FUNCTION_BLOCK FB_Base
VAR_INPUT
END_VAR
VAR_OUTPUT
END_VAR
VAR
	_CalcCounter : INT;
END_VAR

{attribute 'monitoring' := 'call'}
PROPERTY CalcCounter : INT
GET
CalcCounter := _CalcCounter;
END_GET
SET
_CalcCounter := CalcCounter;
END_SET
END_PROPERTY

{attribute 'TcRpcEnable'}
METHOD Calculation : REAL
VAR_INPUT	
	in1, in2 : REAL;
	operator : E_Operator;
END_VAR
CASE operator OF
	E_Operator.idle_operator:
		;
	E_Operator.sum_operator:
		Calculation := in1 + in2;
	E_Operator.diff_operator:
		Calculation := in1 - in2;
	E_Operator.mul_operator:
		Calculation := in1 * in2;
	E_Operator.ratio_operator:
		IF in2 <> 0 THEN
			Calculation := in1 / in2;
		END_IF	
END_CASE
_CalcCounter := _CalcCounter + 1;
END_METHOD

END_FUNCTION_BLOCK

(* stored: Version 1.1.0.1, ProductVersion 3.1.4024.4
   POU FB_Base: Id {a47b3dd3-3c95-4dd3-a852-b40984128896}, SpecialFunc None
   Property CalcCounter: Id {fcd7ee22-aec1-4153-995f-912de616842c}
   Get Get: Id {1488e565-0a32-43b8-9c5a-1a3bdf452a0b}
   Set Set: Id {f2bc713d-a704-42a1-8f54-24d4e3514627}
   Method Calculation: Id {412fe29f-4f1f-4527-b4ec-f067d5c4a43c} *)
